FUNCTION_BLOCK SERVER_10 (* Connect to a CLIENT_10 Block *)
  (* Standard: 61499-2; Description: Copyright (c) 2017 fortiss GmbH This program and the accompanying materials are made available under the terms of the Eclipse Public License 2.0 which is available at https://www.eclipse.org/legal/epl-2.0/ SPDX-License-Identifier: EPL-2.0 *)
  (* Version 3.0, 2025-04-14, Patrick Aigner, changed package *)
  (* Version 1.0, 2017-10-25, Alois Zoitl, fortiss GmbH, initial API and implementation and/or initial documentation *)
  PACKAGE iec61499::net;
  {SET_ATTRIBUTE(eclipse4diac::core::GenericClassName, 'GEN_SERVER')}
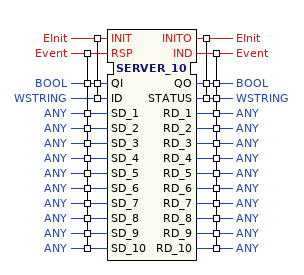
  EVENT_INPUT
    INIT : EInit WITH QI, ID; (* Enable Server for a Client connection (QI = TRUE) / Close Server (QI = FALSE) *)
    RSP WITH QI, SD_1, SD_2, SD_3, SD_4, SD_5, SD_6, SD_7, SD_8, SD_9, SD_10; (* Send data to Client *)
  END_EVENT
  EVENT_OUTPUT
    INITO : EInit WITH QO, STATUS; (* Ready for Client Connection (QI = TRUE) / Closed  (QI = FALSE) *)
    IND WITH QO, STATUS, RD_1, RD_2, RD_3, RD_4, RD_5, RD_6, RD_7, RD_8, RD_9, RD_10; (* New data available from Client *)
  END_EVENT
  VAR_INPUT
    QI : BOOL;
    ID : WSTRING;
    SD_1 : ANY;
    SD_2 : ANY;
    SD_3 : ANY;
    SD_4 : ANY;
    SD_5 : ANY;
    SD_6 : ANY;
    SD_7 : ANY;
    SD_8 : ANY;
    SD_9 : ANY;
    SD_10 : ANY;
  END_VAR
  VAR_OUTPUT
    QO : BOOL;
    STATUS : WSTRING;
    RD_1 : ANY;
    RD_2 : ANY;
    RD_3 : ANY;
    RD_4 : ANY;
    RD_5 : ANY;
    RD_6 : ANY;
    RD_7 : ANY;
    RD_8 : ANY;
    RD_9 : ANY;
    RD_10 : ANY;
  END_VAR
END_FUNCTION_BLOCK
